// TIA Portal V19 export
TYPE "LAF_typeDevDiagInterface"
TITLE = typeDevDiagInterface
// This data type represents the structure of the data block „InstDevDiagInterface“.  
// 
// **PLC Data types**  
// * [LAF_typeDevDiagGlobal](../Library%20Types/LAF_typeDevDiagGlobal.htm)  
// * [LAF_typeDevDiagBasic](../Library%20Types/LAF_typeDevDiagBasic.htm)  
// * [LAF_typeDevDiagState](../Library%20Types/LAF_typeDevDiagState.htm)
// Struktur Profinet device Diagnose
// stored: Access Published
   STRUCT
      globalInfoHmi : "LAF_typeDevDiagGlobal";   // Globale Informationen für HMI PN Device Diag / Global information Profinet device diag HMI
      devStateHmi { ExternalWritable := 'False'} : Array[0..256] of "LAF_typeDevDiagBasic";   // Status Informationen für HMI PN Device Diag / Status information Profinet device diag HMI
      devStateUser { ExternalAccessible := 'False'; ExternalVisible := 'False'; ExternalWritable := 'False'} : Array[0..256] of "LAF_typeDevDiagState";   // Anwender-Schnittstelle Status Device Diag / User interface Profinet device diag
   END_STRUCT;
END_TYPE
